TYPE T_DATA_TYPE : INT; END_TYPE

(* stored: Version 1.1.0.1, ProductVersion 3.1.4024.4
   DUT T_DATA_TYPE: Id {81665eb3-df04-4851-ab82-63315c4b3331} *)
